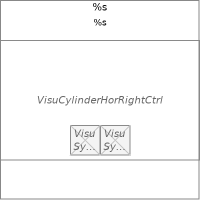
VISUALIZATION VisuCylinderGripperDown  // 200x200
VAR_IN_OUT
	fbVisuCylinder: FB_VISU_CYLINDER;
END_VAR
    Textfield (0,15 200x15), "%s", text variable: fbVisuCylinder.strInfo, colour toggle: fbVisuCylinder.stEvent.bEventActive
    Textfield (0,0 200x14), "%s", text variable: fbVisuCylinder.strFullObjName
    Group (40,40 120x80)
        OnMouseClick: execute { fbVisuCylinder.bFrameInvisible:=false; }
        RoundedRectangle (85,30 20x50)
            p3560616238: fbVisuCylinder.iMoveSmall
        RoundedRectangle (5,30 20x50)
            p3560616238: fbVisuCylinder.iNegMoveSmall
        RoundedRectangle (0,20 110x20)
        Rectangle (0,0 110x45)
    Group (70,125 60x30)
        Image (0,0 30x30), invisible if: fbVisuCylinder.bWorkArrowInvisible, image: VisuSymbols.Symbols.ArrowBoldRight
            p2175578022: fbVisuCylinder.dwFrameColorWork
        Image (30,0 30x30), invisible if: fbVisuCylinder.bWorkArrowInvisible, image: VisuSymbols.Symbols.ArrowBoldLeft
            p2175578022: fbVisuCylinder.dwFrameColorWork
    Group (70,125 60x30)
        Image (0,0 30x30), invisible if: fbVisuCylinder.bBaseArrowInvisible, image: VisuSymbols.Symbols.ArrowBoldLeft
            p2175578022: fbVisuCylinder.dwFrameColorBase
        Image (30,0 30x30), invisible if: fbVisuCylinder.bBaseArrowInvisible, image: VisuSymbols.Symbols.ArrowBoldRight
            p2175578022: fbVisuCylinder.dwFrameColorBase
    Frame (0,40 200x120), invisible if: fbVisuCylinder.bFrameInvisible, frame switch variable: fbVisuCylinder.iFrame
        shows VisuCylinderHorRightCtrl(fbVisuCylinder := fbVisuCylinder)
END_VISUALIZATION

(* stored: Version 1.1.0.1, ProductVersion 3.1.4024.12
   Visu VisuCylinderGripperDown: Id {2c95f386-ca21-4eaf-95e6-b75d44ad8dcc} *)
